PROGRAM ReactorLevelAndPressure
VAR
	_iPressureScaledValue: INT; //Scaled pressure value
	_bLevelControlSwitch : BOOL;
	_slurryInValveCommand : BOOL;
	_slurryOutValveCommand : BOOL;
	_pressureIntervals : ST_PressureIntervals;
	
	levelControlMode : INT;
	manualModeEntered : BOOL;
	autoModeEntered : BOOL;
	SFE_ReactorValveControl: FB_ReactorValves;
	sLevelControlState: STRING;
//	sLevelValveState: STRING;
	sFillingValveState: STRING;
	timeControlToggle: FB_toggleheartbeat;
	
	_extractiveOutOnOffValveCommand : BOOL;
	
	HandleExtractiveOutlet : FB_ExtractiveOutletHandler;
END_VAR
VAR PERSISTENT
	_fillingValveOpenInterval: INT;
	_fillingValveCloseInterval: INT;	
	PressureUpperInterVal_1: INT;
	PressureUpperInterVal_2: INT;
	PressureLowerInterval_1: INT;
	PressureLowerInterval_2: INT;	
	PressureUpperInterVal_3: INT;
	PressureLowerInterval_3: INT;
END_VAR

// Scale analog pressure
_iPressureScaledValue := F_AnalogScale(AnalogInputRawValue := GVL_IO.reactorPressure, MaxAnalogValue := 1000);

IF _bLevelControlSwitch THEN
	levelControlMode := 1;
ELSE
	levelControlMode := 0;
END_IF

// Control logic according to level mode selection
CASE levelControlMode OF
	0:
		//LevelControl.sLevelControlState := 'MAN';
		sLevelControlState := 'MAN';
		// Close inlet/outlet valves when manual mode entered
		IF NOT manualModeEntered THEN
			GVL_IO.reactorInletValve := FALSE; // Close all valves when auto mode is exited
			GVL_IO.reactorOutletValve := FALSE;
			autoModeEntered := FALSE;
			manualModeEntered := TRUE;
		END_IF
		GVL_IO.reactorInletValve := _slurryInValveCommand;
		GVL_IO.reactorOutletValve := _slurryOutValveCommand;
		
	1:
		IF NOT autoModeEntered THEN
			GVL_IO.reactorInletValve := TRUE; // Open inlet valve when auto mode is entered
			manualModeEntered := FALSE;
			autoModeEntered := TRUE;
		END_IF
		//LevelControl.sLevelControlState := 'AUTO';
		sLevelControlState := 'AUTO';
		
		// Reactor inlet valve: auto control according to timed intervals:
		SFE_ReactorValveControl.onOffTimeControl(
										openInterValSecs := _fillingValveOpenInterval,
										closeIntervalSecs := _fillingValveCloseInterval,
										);
		GVL_IO.reactorInletValve := SFE_ReactorValveControl.timeControlOpen;
		// Reactor outlet valve: auto control according to pressure intervals
		SFE_ReactorValveControl.pressureIntervalControl(
												interval_1_condition:= GVL_IO.reactorLevelHigh AND GVL_IO.reactorInletValve, // If above higher limit and filling valve open
												pressureUpperInterval_1:= _pressureIntervals.PressureUpperInterval_1, 
												pressureLowerInterval_1:= _pressureIntervals.PressureLowerInterval_1, 
												interval_2_condition:= GVL_IO.reactorLevelHigh AND NOT GVL_IO.reactorInletValve,  // If above higher limit and filling valve closed
												pressureUpperInterval_2:= _pressureIntervals.PressureUpperInterval_2, 
												pressureLowerInterval_2:= _pressureIntervals.PressureLowerInterval_2, 
												interval_3_condition:= NOT GVL_IO.reactorLevelHigh AND GVL_IO.reactorInletValve,  // If below higher limit and reactor filling valve open
												pressureUpperInterval_3:= _pressureIntervals.PressureUpperInterval_3, 
												pressureLowerInterval_3:= _pressureIntervals.PressureLowerInterval_3, 
												pressureValue:= _iPressureScaledValue, 
												pressureReference:= DINT_TO_INT(SerialCommunicationHandler.pumpingPressureSetpoint), 
												valveOpenCondition:= NOT (NOT GVL_IO.reactorLevelHigh AND NOT GVL_IO.reactorInletValve), 
												forceValveClosed:= (NOT GVL_IO.reactorLevelHigh AND NOT GVL_IO.reactorInletValve),
												);
		GVL_IO.reactorOutletValve := SFE_ReactorValveControl.pressureControlOpen;
END_CASE

timeControlToggle(I_OpenInterValSecs := 5, I_CloseIntervalSecs := 10, O_Update => );

// Extractive outlet control
HandleExtractiveOutlet(
					onOffValveCommand := _extractiveOutOnOffValveCommand,
					onOffValveOpen => GVL_IO.extractiveOutletOnOffValve);

PROPERTY bLevelControlSwitch : BOOL
SET

_bLevelControlSwitch := bLevelControlSwitch;
END_SET
END_PROPERTY

PROPERTY ExtractiveOutOnOffValveCommand : BOOL
SET

_extractiveOutOnOffValveCommand := ExtractiveOutOnOffValveCommand;
END_SET
END_PROPERTY

PROPERTY fillingValveCloseInterval : INT
SET

_fillingValveCloseInterval := fillingValveCloseInterval;
END_SET
END_PROPERTY

PROPERTY fillingValveOpenInterval : INT
SET

_fillingValveOpenInterval := fillingValveOpenInterval;
END_SET
END_PROPERTY

PROPERTY iPressureScaledValue : INT
GET

iPressureScaledValue := _iPressureScaledValue;
END_GET
END_PROPERTY

PROPERTY PressureIntervals : ST_PressureIntervals
SET

_pressureIntervals := PressureIntervals;
END_SET
END_PROPERTY

PROPERTY SlurryInValveCommand : BOOL
SET

_slurryInValveCommand := SlurryInValveCommand;
END_SET
END_PROPERTY

PROPERTY SlurryOutValveCommand : BOOL
SET

_slurryOutValveCommand := SlurryOutValveCommand;
END_SET
END_PROPERTY

END_PROGRAM

(* stored: Version 1.1.0.1, ProductVersion 3.1.4024.9
   POU ReactorLevelAndPressure: Id {a387b85d-f129-4119-abd4-456930450f01}, SpecialFunc None
   Property bLevelControlSwitch: Id {157d05c6-890c-4007-9267-879a33c29919}
   Set Set: Id {6f409d45-6c86-41c4-88fa-9adadc01cff5}
   Property ExtractiveOutOnOffValveCommand: Id {461a6a9f-281d-484c-948f-8a31cb53f17c}
   Set Set: Id {56f473f2-6b90-480e-9099-0f83e1c5bbdc}
   Property fillingValveCloseInterval: Id {6a88157e-ad1e-4b33-b420-23e077b392b3}
   Set Set: Id {ecae8a8d-2f82-4ab1-b797-5f8a6ba22e3e}
   Property fillingValveOpenInterval: Id {1a5a0701-ed7c-4ad0-b561-bf5a253bdcbd}
   Set Set: Id {c5a68f5f-e948-4258-ab24-2caf6453de2b}
   Property iPressureScaledValue: Id {f3fccc10-a324-4a46-aa67-2f5a5ade620e}
   Get Get: Id {b24340e3-e276-44cc-aedf-92fb116f5053}
   Property PressureIntervals: Id {590fbcd9-9ded-465e-b5f3-c87f976ee592}
   Set Set: Id {55337214-2fb9-445e-aa8b-e3a09f5ae5e0}
   Property SlurryInValveCommand: Id {cf2e99f8-1ae2-4412-8aaa-3a3f4953daac}
   Set Set: Id {fa7013a0-5634-4bfb-bf36-3d02e0323469}
   Property SlurryOutValveCommand: Id {28697755-784a-4676-838b-2343170d2384}
   Set Set: Id {b5d4a71f-8119-4ac2-95c8-c61337f36845} *)
